// TIA Portal V20 export
DATA_BLOCK "ET500SP_507"   // DB236
// stored: MemoryReserve 100
   VAR
      "SP507.00 ELECTRODE NG KICKER DETECT SENSOR" : Bool;
      "SP507.01 ELECTRODE DETECT COLOR SENSOR #1" : Bool;
      "SP507.02 ELECTRODE DETECT COLOR SENSOR #2" : Bool;
      SPARE1 : Bool;
      "SP507.04 OutputCam_PassKickerAxisZ" : Bool;
      SPARE2 : Bool;
      SPARE3 : Bool;
      SPARE4 : Bool;
      SPARE5 : Bool;
   END_VAR
BEGIN
END_DATA_BLOCK
